FUNCTION F_ADD_REF_F : BOOL
VAR_IN_OUT
	fValueRoot	: LREAL;
END_VAR
VAR_INPUT
	fValue		: LREAL;
END_VAR

fValueRoot := fValueRoot + fValue;

END_FUNCTION

(* stored: Version 1.1.0.1, ProductVersion 3.1.4024.12
   POU F_ADD_REF_F: Id {52e63c61-d602-454e-98d8-f10302fc4063}, SpecialFunc None *)
